(* PLC project trend, Dassault Systèmes ControlBuild 2024x *)
(* stored: creationDateTime 2023-10-03T11:13:25-01:00 *)

(* This module simulates the evolution of a measure in function of the time. The operator can simulate a "ax + b" curve . *)
FUNCTION_BLOCK equipment_library.trend
  VAR_INPUT
    gradient : REAL := 0.0;
    interceptPoint : REAL := 0.0;
  END_VAR
  VAR_OUTPUT
    A : REAL := 0.0;
    B : REAL := 0.0;
    time : REAL := 0.0;
    realOutput : REAL := 0.0;
    theoricalOutput : REAL := 0.0;
  END_VAR
  VAR
    memoSlope : REAL := 0.0;
    memoInc : REAL := 0.0;
  END_VAR
  VAR
    d_resetParameters : BOOL := false;
    v_d_resetParameters : BOOL := false;
    d_intermediatePresetting : BOOL := false;
    v_d_intermediatePresetting : REAL := 0.0;
  END_VAR


ACTION C_source_code:
/* ----------------------------------------------------------------	*/
/* Type : Model of Operative Behaviour					*/
/* Category :  Toolbox							*/
/* Author : Dassault Systemes						*/
/* Update date : June 2018						*/
/* ----------------------------------------------------------------	*/
/* This module simulates the addition of two real numbers.		*/
/* ----------------------------------------------------------------	*/
/* This module simulates the evolution of a measure in function of 	*/
/* the time. The operator can simulate a "ax + b" curve .		*/
/* Nota :									*/
/*	- an action on the gradient changes the slope while keeping  	*/
/*		continuity.							*/
/*	- an action on intercept point keeps the slope and force 	*/
/*		only intercept point.					*/
/*	- the time variable is reinitialized at each gradient		*/
/*		or intercept point change. 					*/
/* ----------------------------------------------------------------	*/

if (d_resetParameters) {
	realOutput=0;
	theoricalOutput=0;
	A=0;
	B=0;
	time=0;
	memoSlope=0;
	memoInc=0;
}
else {
	if (gradient != memoSlope) {
		memoSlope = gradient;
		A=gradient;
		B=theoricalOutput;
		time=0;
	}
	if (interceptPoint != memoInc) {
		memoInc=interceptPoint;
		B=interceptPoint;
		time=0;
	}
	time=time+(CLOCK_PERIOD/1000000);
	theoricalOutput=A*time+B;

	if (d_intermediatePresetting) 
		realOutput=v_d_intermediatePresetting;
	else 
		realOutput=theoricalOutput;
}
END_ACTION
END_FUNCTION_BLOCK
